(* IEC 61131-3 sources: XPGAnalyser/bac/Armoire_Gaz/ihm/scripts, 7 files *)

(* ---- 0070-Suivi_Maintenance.st ---- *)
IF Mode_Maintenance THEN
    Message_Operateur := 'Maintenance en cours';
    IHM_JOURNAL('Passage en maintenance');
ELSE
    Message_Operateur := 'Production';
    IHM_JOURNAL('Retour en production');
END_IF;

(* ---- 0154-Statistiques_Pression.st ---- *)
(* Mini et maxi de la pression A, depuis le lancement de l'IHM *)
VAR
    Mini : REAL := 1000.0;   (* VAR : gardée d'une exécution à l'autre *)
    Maxi : REAL;
    Tours : DINT;
    Ecart : REAL;
END_VAR
VAR_TEMP
    P : REAL;                (* VAR_TEMP : repart à chaque exécution *)
END_VAR

P := Armoires[0].ana.PT1.mes;
Tours := Tours + 1;
IF P < Mini THEN
    Mini := P;
END_IF;
IF P > Maxi THEN
    Maxi := P;
END_IF;
IF Tours MOD 5 = 0 THEN
    IHM_JOURNAL('Pression A : mini {Mini:0.0}, maxi {Maxi:0.0} bar ({Tours} mesures)');
END_IF;
IF Moyenne_Pression(P, Armoires[1].ana.PT1.mes) > 30.0 THEN
    Tracer_Evenement('Moyenne haute', 2);
END_IF;

(* ---- 0228-Passage_Nuit.st ---- *)
(* Le mode nuit : la vue des commandes s'assombrit, le programmateur s'efface *)
IF Mode_Nuit THEN
    Vue_Commandes.Background := '#0B0F14';
    Vue_Commandes.Prog_Chauffage.Visible := FALSE;
    Vue_Commandes.Inter_Pompe.ColorOn := '#F2994A';
    Vue_Commandes.Titre_Commandes.Text := 'Pompe de transfert : mode nuit';
    Vue_Commandes.Texte_Valeurs.TextColor := '#F2C94C';
ELSE
    Vue_Commandes.Background := '#20242B';
    Vue_Commandes.Prog_Chauffage.Visible := TRUE;
    Vue_Commandes.Inter_Pompe.ColorOn := '#2ECC71';
    Vue_Commandes.Titre_Commandes.Text := 'Pompe de transfert : commandes';
    Vue_Commandes.Texte_Valeurs.TextColor := '#9CC3E6';
END_IF;
IHM_JOURNAL('Mode nuit {Mode_Nuit:activé|désactivé} par {SYS.UserName} à {SYS.Time}');

(* ---- 0241-Animation_Ligne.st ---- *)
(* Les mesures de la ligne de gaz, simulees toutes les 100 ms *)
Temps_Ligne := Temps_Ligne + 0.1;
(* L'essai de surpression : la pression monte tant qu'on appuie *)
IF Essai_Surpression AND Surpression < 6.0 THEN
    Surpression := Surpression + 0.3;
ELSIF NOT Essai_Surpression AND Surpression > 0.0 THEN
    Surpression := Surpression - 0.3;
END_IF;
Pression_Ligne := 8.0 + 2.0 * SIN(Temps_Ligne * 0.3) + Surpression;
Temperature_Local := 21.0 + 3.0 * SIN(Temps_Ligne * 0.05);
Niveau_Cuve := 60.0 + 30.0 * SIN(Temps_Ligne * 0.15);
IF Pompe_Marche THEN
    Debit_Ligne := 120.0 + 20.0 * SIN(Temps_Ligne * 0.4);
    Pieces_Produites := Pieces_Produites + 1.0;
ELSE
    Debit_Ligne := Debit_Ligne * 0.9;
END_IF;
(* L'etat de la pompe : en defaut au-dessus de 13 bar *)
IF Pression_Ligne > 13.0 THEN
    Etat_Pompe := 2;
ELSIF Pompe_Marche THEN
    Etat_Pompe := 1;
ELSE
    Etat_Pompe := 0;
END_IF;

(* ---- 0271-Animation_Synoptique.st ---- *)
(* La vue synoptique : le verin va et vient, le silo se vide dans la tremie *)
Temps_Synoptique := Temps_Synoptique + 0.1;
Position_Verin := 50.0 - 50.0 * COS(Temps_Synoptique * 0.8);
IF Marche_Ligne THEN
    Niveau_Silo := Niveau_Silo - 0.25;
    Charge_Tremie := Charge_Tremie + 0.35;
END_IF;
IF Niveau_Silo < 15.0 THEN
    Niveau_Silo := 90.0;
END_IF;
IF Charge_Tremie > 90.0 THEN
    Charge_Tremie := 20.0;
END_IF;

(* ---- 0381-Production_Ligne.st ---- *)
(* La ligne 1 : 2,5 pieces par seconde quand la pompe tourne, un rebut sur treize *)
IF Pompe_Marche THEN
    Fraction_Piece := Fraction_Piece + 0.25;
END_IF;
IF Fraction_Piece >= 1.0 THEN
    Fraction_Piece := Fraction_Piece - 1.0;
    IF ((Pieces_Bonnes + Rebuts_Ligne) MOD 13) = 12 THEN
        Rebuts_Ligne := Rebuts_Ligne + 1;
    ELSE
        Pieces_Bonnes := Pieces_Bonnes + 1;
    END_IF;
END_IF;

(* ---- 0622-Surveillance_Fours.st ---- *)
VAR
    i : INT;
    f : INT;
    somme : REAL;
END_VAR
(* Surveillance des fours : la moyenne des consignes, les fours trop chauds *)
somme := 0.0;
FOR i := Consignes.Low TO Consignes.High DO
    somme := somme + Consignes[i];
END_FOR;
FOR f := 1 TO Fours.High DO
    IF Fours[f].Temperature > Fours[f].Consigne + 20.0 THEN
        Fours[f].Vannes[1].Position := 0;
        IHM_JOURNAL('Four {f} trop chaud');
    END_IF;
END_FOR;
